// TIA Portal V19 export
DATA_BLOCK "EmNodes"   // DB42
// stored: Access Published, MemoryReserve 100, Namespace Unit2
   VAR
      unitStatus { ExternalWritable := 'False'} : "LAF_typeUnitStatus";   // Status of the unit
      emFeedback { ExternalWritable := 'False'} : Array[0.._.Unit2_NO_OF_EMs] of "LUC_typeEmFeedback";   // Status of the individual equipment modules
      emRelations { ExternalWritable := 'False'} : Struct   // This is an example
         EM1 { S7_SetPoint := 'True'} : "LEXCHANGETRAY_typeRoller_interface";
         EM2 : "LEXCHANGETRAY_typeConstraintRollerEm_interface";
         EM3 { S7_SetPoint := 'True'} : "LEXCHANGETRAY_typeConstraintWorkstationEm_interface";
         EM6 : "LEXCHANGETRAY_typeRoller_interface_B2";
         EM5 : "LEXCHANGETRAY_typePlasticEm5_interface";
         EM4 : "LEXCHANGETRAY_typeHandlingXyzEm_interface";
      END_STRUCT;
      signalStack { ExternalWritable := 'False'} : "LUC_typeSignalStackByBool";
      actionEmManager { S7_SetPoint := 'True'} : "LEXCHANGETRAY_typeEmActionManager";
      emStatus : Array[0.._.Unit2_NO_OF_EMs] of "LUC_typeStates";
   END_VAR
BEGIN
END_DATA_BLOCK
